FUNCTION_BLOCK FB_LamparaConmutada_SFC
VAR_INPUT
END_VAR
VAR_OUTPUT
END_VAR
VAR
    Lampara AT %Q*: BOOL;
    Pulsador AT %I*: BOOL;
    
    Pulsacion: Tc2_Standard.R_TRIG;
END_VAR

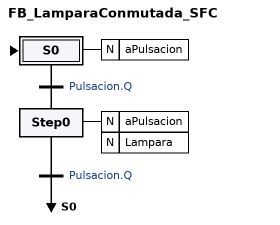
INITIAL_STEP S0:
    aPulsacion(N);
END_STEP
TRANSITION FROM S0 TO Step0
    := Pulsacion.Q;
END_TRANSITION
STEP Step0:
    aPulsacion(N);
    Lampara(N);
END_STEP
TRANSITION FROM Step0 TO S0
    := Pulsacion.Q;
END_TRANSITION

ACTION aPulsacion:
Pulsacion(CLK := Pulsador);
END_ACTION

END_FUNCTION_BLOCK

(* stored: Version 1.1.0.1, ProductVersion 3.1.4024.12
   POU FB_LamparaConmutada_SFC: Id {627d8519-ef3d-4358-89ad-fa30f84c70ba}, SpecialFunc None
   Action aPulsacion: Id {692c89e8-9cde-44df-ba38-bfdc617d6826} *)
